// TIA Portal V18 export
TYPE "UDT_settingsShift"
   STRUCT
      shiftEN { ExternalVisible := 'False'} : DInt;
      shiftBegin { ExternalVisible := 'False'} : Time_Of_Day;
      shiftEnd { ExternalVisible := 'False'} : Time_Of_Day;
      break1EN { ExternalVisible := 'False'} : DInt;
      break1Begin { ExternalVisible := 'False'} : Time_Of_Day;
      break1End { ExternalVisible := 'False'} : Time_Of_Day;
      break2EN { ExternalVisible := 'False'} : DInt;
      break2Begin { ExternalVisible := 'False'} : Time_Of_Day;
      break2End { ExternalVisible := 'False'} : Time_Of_Day;
      break3EN { ExternalVisible := 'False'} : DInt;
      break3Begin { ExternalVisible := 'False'} : Time_Of_Day;
      break3End { ExternalVisible := 'False'} : Time_Of_Day;
      break4EN { ExternalVisible := 'False'} : DInt;
      break4Begin { ExternalVisible := 'False'} : Time_Of_Day;
      break4End { ExternalVisible := 'False'} : Time_Of_Day;
      break5EN { ExternalVisible := 'False'} : DInt;
      break5Begin { ExternalVisible := 'False'} : Time_Of_Day;
      break5End { ExternalVisible := 'False'} : Time_Of_Day;
      targetEN { ExternalVisible := 'False'} : DInt;
      target { ExternalVisible := 'False'} : DInt;
      taktTimeEN { ExternalVisible := 'False'} : DInt;
      taktTime { ExternalVisible := 'False'} : DInt;
   END_STRUCT;
END_TYPE
